// TIA Portal V19 export
DATA_BLOCK "DB_ALGORYTHM"   // DB4
// stored: InstanceOfName FB_ALGORYTHM, InstanceOfType FB
"FB_ALGORYTHM"
   // VAR_IN_OUT
   //    FB_CONVEYOR1_DB : "FB_CONVEYOR";
   //    FB_COVEYOR2_DB : "FB_CONVEYOR";
   //    FB_COVEYOR3_DB : "FB_CONVEYOR";
   //    FB_COVEYOR4_DB : "FB_CONVEYOR";
   //    FB_COVEYOR5_DB : "FB_CONVEYOR";
   //    FB_COVEYOR6_DB : "FB_CONVEYOR";
   //    FB_COVEYOR7_DB : "FB_CONVEYOR";
   //    FB_COVEYOR8_DB : "FB_CONVEYOR";
   //    FB_COVEYOR9_DB : "FB_CONVEYOR";
   //    FB_COVEYOR10_DB : "FB_CONVEYOR";
   //    dtShifter1_DB : "Shifter_DT";
   //    dtShifter2_DB : "Shifter_DT";
   //    dtShifter3_DB : "Shifter_DT";
   //    dtShifter4_DB : "Shifter_DT";
   //    dtShifter5_DB : "Shifter_DT";
   //    dtEntryConveyor_DB : "Entry_conveyor";
   //    dtDataBlock_DB : "Data_Block";
   // END_VAR
BEGIN
END_DATA_BLOCK
